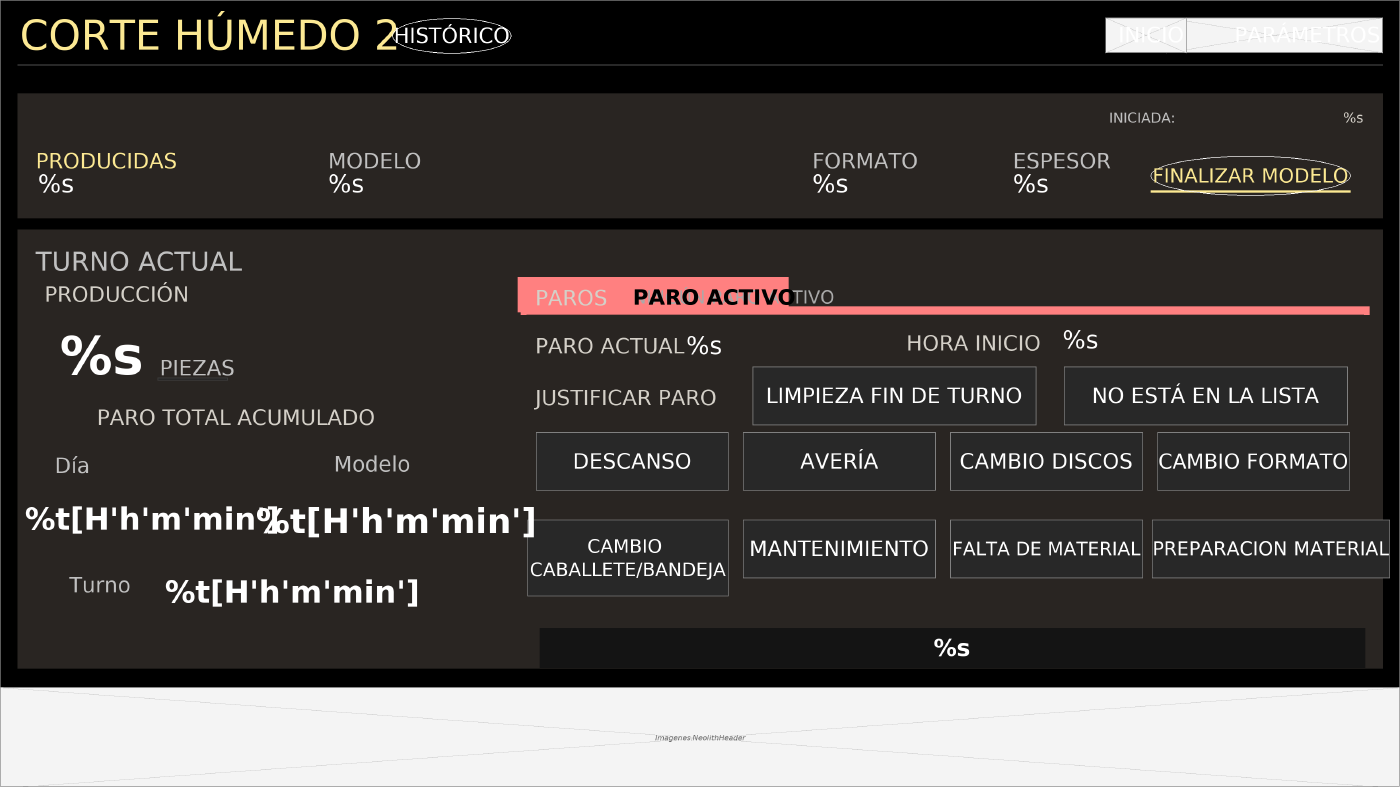
VISUALIZATION Home_CortH2  // 1920x1080
    Rectangle (24,315 1872x602)
    Rectangle (24,128 1872x171)
    Rectangle (24,88 1872x2)
    Label (24,16 514x64), "CORTE HÚMEDO 2"
    Rectangle (1454,451 375x30), "%s", text variable: FuncParoNodoRemote1CorteH2.Funci_CortHum2.H_InParo_Ftc, invisible if: FuncParoNodoRemote1CorteH2.Funci_CortHum2.M_SinParo_Ftc
    Rectangle (938,459 287x30), "%s", text variable: FuncParoNodoRemote1CorteH2.Funci_CortHum2.Min_Parado_Ftc, invisible if: FuncParoNodoRemote1CorteH2.Funci_CortHum2.M_SinParo_Ftc
    Rectangle (1573,147 300x30), "%s", text variable: FuncParoNodoRemote1CorteH2.sFechaInicModeloTab
    Label (1518,147 99x30), "INICIADA:"
    Rectangle (740,862 1132x54), "%s", text variable: FuncParoNodoRemote1CorteH2.Funci_CortHum2.S_Justi_Paro_Ftc, invisible if: FuncParoNodoRemote1CorteH2.Funci_CortHum2.M_SinParo_Ftc, input disabled if: FuncParoNodoRemote1CorteH2.FunGeneCortHum2.IndexJustificacionParo<>10
        OnMouseDown: write the text variable via Edit
    Image (116,-391 250x250), invisible if: FuncParoNodoRemote1CorteH2.Funci_CortHum2.M_SinParo_Ftc, image: ImagePool.Exclamación
    Image (454,-421 250x250), invisible if: FuncParoNodoRemote1CorteH2.Funci_CortHum2.M_SinParo_Ftc, image: ImagePool.Exclamación
    Image (1128,-383 250x250), invisible if: FuncParoNodoRemote1CorteH2.Funci_CortHum2.M_SinParo_Ftc, image: ImagePool.Exclamación
    Image (123,-961 250x250), invisible if: FuncParoNodoRemote1CorteH2.Funci_CortHum2.M_SinParo_Ftc, image: ImagePool.Exclamación
    Image (1136,-683 250x250), invisible if: FuncParoNodoRemote1CorteH2.Funci_CortHum2.M_SinParo_Ftc, image: ImagePool.Exclamación
    Image (478,-696 250x250), invisible if: FuncParoNodoRemote1CorteH2.Funci_CortHum2.M_SinParo_Ftc, image: ImagePool.Exclamación
    Image (1691,-991 250x250), invisible if: FuncParoNodoRemote1CorteH2.Funci_CortHum2.M_SinParo_Ftc, image: ImagePool.Exclamación
    Image (1600,24 296x48), "PARÁMETROS"
        OnMouseClick: change screen: Ajustes_CorteH2
    Image (1516,24 111x48), "INICIO"
        OnMouseClick: change screen: Home_Sel_Maq
    Group (447,203 1095x69)
        Rectangle (0,29 671x40), "%s", text variable: FuncParoNodoRemote1CorteH2.sModeloActualTabla
        Rectangle (939,29 120x40), "%s", text variable: FuncParoNodoRemote1CorteH2.sEspesorActualTabla
        Rectangle (664,29 321x40), "%s", text variable: FuncParoNodoRemote1CorteH2.sFormatoActualTabla
        Label (0,0 487x36), "MODELO"
        Label (664,0 156x36), "FORMATO"
        Label (939,0 156x36), "ESPESOR"
    Label (46,203 199x36), "PRODUCIDAS"
    Rectangle (49,232 248x40), "%s", text variable: FuncParoNodoRemote1CorteH2.Funci_CortHum2.Cont_Piezas_Ftc
    Group (1578,214 274x54)
        Rectangle (0,47 274x3)
        Ellipse (0,0 274x54), "FINALIZAR MODELO"
            OnMouseClick: OpenDialog Dialog=V_Emerg_Fin_Prod_Ch2, OpenModal=True, OpenCentered=True
    Label (46,332 390x54), "TURNO ACTUAL"
    Label (58,386 199x36), "PRODUCCIÓN"
    Label (731,457 261x36), "PARO ACTUAL", invisible if: FuncParoNodoRemote1CorteH2.Funci_CortHum2.M_SinParo_Ftc
    Label (1240,453 261x36), "HORA INICIO", invisible if: FuncParoNodoRemote1CorteH2.Funci_CortHum2.M_SinParo_Ftc
    RoundedRectangle (735,593 264x80), "DESCANSO", invisible if: FuncParoNodoRemote1CorteH2.Funci_CortHum2.M_SinParo_Ftc
        OnMouseClick: execute { FuncParoNodoRemote1CorteH2.FunGeneCortHum2.IndexJustificacionParo:=1; FuncParoNodoRemote1CorteH2.FunGeneCortHum2.ListadoJustificacionParo(); }
    RoundedRectangle (1019,593 264x80), "AVERÍA", invisible if: FuncParoNodoRemote1CorteH2.Funci_CortHum2.M_SinParo_Ftc
        OnMouseClick: execute { FuncParoNodoRemote1CorteH2.FunGeneCortHum2.IndexJustificacionParo:=2; FuncParoNodoRemote1CorteH2.FunGeneCortHum2.ListadoJustificacionParo(); }
    RoundedRectangle (1303,593 264x80), "CAMBIO DISCOS", invisible if: FuncParoNodoRemote1CorteH2.Funci_CortHum2.M_SinParo_Ftc
        OnMouseClick: execute { FuncParoNodoRemote1CorteH2.FunGeneCortHum2.IndexJustificacionParo:=3; FuncParoNodoRemote1CorteH2.FunGeneCortHum2.ListadoJustificacionParo(); }
    RoundedRectangle (1587,593 264x80), "CAMBIO FORMATO", invisible if: FuncParoNodoRemote1CorteH2.Funci_CortHum2.M_SinParo_Ftc
        OnMouseClick: execute { FuncParoNodoRemote1CorteH2.FunGeneCortHum2.IndexJustificacionParo:=4; FuncParoNodoRemote1CorteH2.FunGeneCortHum2.ListadoJustificacionParo(); }
    Rectangle (79,444 183x88), "%s", text variable: FuncParoNodoRemote1CorteH2.Funci_CortHum2.Cont_Piezas_Ftc
    Label (216,487 106x36), "PIEZAS"
    Rectangle (216,518 96x4), colour toggle: FuncParoNodoRemote1CorteH2.Funci_CortHum2.Fotocelula
    Label (731,528 261x36), "JUSTIFICAR PARO", invisible if: FuncParoNodoRemote1CorteH2.Funci_CortHum2.M_SinParo_Ftc
    Rectangle (714,424 1164x4), invisible if: FuncParoNodoRemote1CorteH2.Funci_CortHum2.M_SinParo_Ftc
    Rectangle (710,380 371x48), invisible if: FuncParoNodoRemote1CorteH2.Funci_CortHum2.M_SinParo_Ftc
    Label (731,391 199x36), "PAROS", invisible if: FuncParoNodoRemote1CorteH2.Funci_CortHum2.M_SinParo_Ftc
    Label (865,393 326x30), "NINGÚN PARO ACTIVO", invisible if: FuncParoNodoRemote1CorteH2.Funci_CortHum2.MParo_Ftc
    Label (865,393 235x30), "PARO ACTIVO", invisible if: FuncParoNodoRemote1CorteH2.Funci_CortHum2.M_SinParo_Ftc
    Ellipse (538,25 163x48), "HISTÓRICO"
        OnMouseClick: change screen: HistTablaTablas_Ch2
    Label (130,555 367x36), "PARO TOTAL ACUMULADO"
    Image (-3,943 1927x139), image: Imagenes.NeolithHeader
    RoundedRectangle (723,713 276x105), "CAMBIO CABALLETE/BANDEJA", invisible if: FuncParoNodoRemote1CorteH2.Funci_CortHum2.M_SinParo_Ftc
        OnMouseClick: execute { FuncParoNodoRemote1CorteH2.FunGeneCortHum2.IndexJustificacionParo:=5; FuncParoNodoRemote1CorteH2.FunGeneCortHum2.ListadoJustificacionParo(); }
    RoundedRectangle (1019,713 264x80), "MANTENIMIENTO", invisible if: FuncParoNodoRemote1CorteH2.Funci_CortHum2.M_SinParo_Ftc
        OnMouseClick: execute { FuncParoNodoRemote1CorteH2.FunGeneCortHum2.IndexJustificacionParo:=6; FuncParoNodoRemote1CorteH2.FunGeneCortHum2.ListadoJustificacionParo(); }
    RoundedRectangle (1303,713 264x80), "FALTA DE MATERIAL", invisible if: FuncParoNodoRemote1CorteH2.Funci_CortHum2.M_SinParo_Ftc
        OnMouseClick: execute { FuncParoNodoRemote1CorteH2.FunGeneCortHum2.IndexJustificacionParo:=7; FuncParoNodoRemote1CorteH2.FunGeneCortHum2.ListadoJustificacionParo(); }
    RoundedRectangle (1580,713 326x80), "PREPARACION MATERIAL", invisible if: FuncParoNodoRemote1CorteH2.Funci_CortHum2.M_SinParo_Ftc
        OnMouseClick: execute { FuncParoNodoRemote1CorteH2.FunGeneCortHum2.IndexJustificacionParo:=8; FuncParoNodoRemote1CorteH2.FunGeneCortHum2.ListadoJustificacionParo(); }
    RoundedRectangle (1032,503 389x80), "LIMPIEZA FIN DE TURNO", invisible if: FuncParoNodoRemote1CorteH2.Funci_CortHum2.M_SinParo_Ftc
        OnMouseClick: execute { FuncParoNodoRemote1CorteH2.FunGeneCortHum2.IndexJustificacionParo:=9; FuncParoNodoRemote1CorteH2.FunGeneCortHum2.ListadoJustificacionParo(); }
    RoundedRectangle (1459,503 389x80), "NO ESTÁ EN LA LISTA", invisible if: FuncParoNodoRemote1CorteH2.Funci_CortHum2.M_SinParo_Ftc
        OnMouseClick: execute { FuncParoNodoRemote1CorteH2.FunGeneCortHum2.IndexJustificacionParo:=10; FuncParoNodoRemote1CorteH2.FunGeneCortHum2.ListadoJustificacionParo(); }
    Rectangle (31,668 295x88), "%t[H'h'm'min']", text variable: FuncParoNodoRemote1CorteH2.Funci_CortHum2.fbTiempParoAcumDiario.t_Acumulado
    Label (72,621 76x36), "Día"
    Rectangle (223,768 325x88), "%t[H'h'm'min']", text variable: FuncParoNodoRemote1CorteH2.Funci_CortHum2.fbTiempParoAcumTurno.t_Acumulado
    Label (92,785 102x36), "Turno"
    Rectangle (348,671 388x88), "%t[H'h'm'min']", text variable: FuncParoNodoRemote1CorteH2.Funci_CortHum2.fbTiempParoAcumModelo.t_Acumulado
    Label (455,619 118x36), "Modelo"
END_VISUALIZATION

(* stored: Version 1.1.0.1, ProductVersion 3.1.4024.12
   Visu Home_CortH2: Id {f7a066aa-51fa-41a5-a125-f7a911912ae5} *)
